TYPE ST_Log :
STRUCT
	tTime: TIME;
	sCompletion: STRING;
	stTargetLED: ST_LED;
	tET: TIME;
END_STRUCT
END_TYPE

(* stored: Version 1.1.0.1, ProductVersion 3.1.4022.12
   DUT ST_Log: Id {e8a01d42-1619-4507-ab5f-483454a2bd02} *)
